DATA_BLOCK "DB_Z200_HMI"
{ DB_Accessible_From_OPC_UA := 'FALSE' ;
 DB_Accessible_From_Webserver := 'FALSE' ;
 S7_Optimized_Access := 'FALSE' }
VERSION : 0.1
NON_RETAIN
   STRUCT
      tALM { ExternalWritable := 'False'} : Struct   // HMI Alarms
         tE { ExternalWritable := 'False'} : Struct   // Emergency alarms
            xSpare_0 { ExternalWritable := 'False'} : Bool;
            xSpare_1 { ExternalWritable := 'False'} : Bool;
            xSpare_2 { ExternalWritable := 'False'} : Bool;
            xSpare_3 { ExternalWritable := 'False'} : Bool;
            xSpare_4 { ExternalWritable := 'False'} : Bool;
            xSpare_5 { ExternalWritable := 'False'} : Bool;
            xSpare_6 { ExternalWritable := 'False'} : Bool;
            xSpare_7 { ExternalWritable := 'False'} : Bool;
            xSpare_8 { ExternalWritable := 'False'} : Bool;
            xSpare_9 { ExternalWritable := 'False'} : Bool;
            xSpare_10 { ExternalWritable := 'False'} : Bool;
            xSpare_11 { ExternalWritable := 'False'} : Bool;
            xSpare_12 { ExternalWritable := 'False'} : Bool;
            xSpare_13 { ExternalWritable := 'False'} : Bool;
            xSpare_14 { ExternalWritable := 'False'} : Bool;
            xSpare_15 { ExternalWritable := 'False'} : Bool;
            xSpare_16 { ExternalWritable := 'False'} : Bool;
            xSpare_17 { ExternalWritable := 'False'} : Bool;
            xSpare_18 { ExternalWritable := 'False'} : Bool;
            xSpare_19 { ExternalWritable := 'False'} : Bool;
            xSpare_20 { ExternalWritable := 'False'} : Bool;
            xSpare_21 { ExternalWritable := 'False'} : Bool;
            xSpare_22 { ExternalWritable := 'False'} : Bool;
            xSpare_23 { ExternalWritable := 'False'} : Bool;
            xSpare_24 { ExternalWritable := 'False'} : Bool;
            xSpare_25 { ExternalWritable := 'False'} : Bool;
            xSpare_26 { ExternalWritable := 'False'} : Bool;
            xSpare_27 { ExternalWritable := 'False'} : Bool;
            xSpare_28 { ExternalWritable := 'False'} : Bool;
            xSpare_29 { ExternalWritable := 'False'} : Bool;
            xSpare_30 { ExternalWritable := 'False'} : Bool;
            xSpare_31 { ExternalWritable := 'False'} : Bool;
         END_STRUCT;
         tS { ExternalWritable := 'False'} : Struct   // Stopping faults
            xSpare_0 { ExternalWritable := 'False'} : Bool;   //
            xSpare_1 { ExternalWritable := 'False'} : Bool;
            xSpare_2 { ExternalWritable := 'False'} : Bool;
            xSpare_3 { ExternalWritable := 'False'} : Bool;
            xSpare_4 { ExternalWritable := 'False'} : Bool;
            xSpare_5 { ExternalWritable := 'False'} : Bool;
            xSpare_6 { ExternalWritable := 'False'} : Bool;
            xSpare_7 { ExternalWritable := 'False'} : Bool;
            xSpare_8 { ExternalWritable := 'False'} : Bool;
            xSpare_9 { ExternalWritable := 'False'} : Bool;
            xSpare_10 { ExternalWritable := 'False'} : Bool;
            xSpare_11 { ExternalWritable := 'False'} : Bool;
            xSpare_12 { ExternalWritable := 'False'} : Bool;
            xSpare_13 { ExternalWritable := 'False'} : Bool;
            xSpare_14 { ExternalWritable := 'False'} : Bool;
            xSpare_15 { ExternalWritable := 'False'} : Bool;
            xSpare_16 { ExternalWritable := 'False'} : Bool;
            xSpare_17 { ExternalWritable := 'False'} : Bool;
            xSpare_18 { ExternalWritable := 'False'} : Bool;
            xSpare_19 { ExternalWritable := 'False'} : Bool;
            xSpare_20 { ExternalWritable := 'False'} : Bool;
            xSpare_21 { ExternalWritable := 'False'} : Bool;
            xSpare_22 { ExternalWritable := 'False'} : Bool;
            xSpare_23 { ExternalWritable := 'False'} : Bool;
            xSpare_24 { ExternalWritable := 'False'} : Bool;
            xSpare_25 { ExternalWritable := 'False'} : Bool;
            xSpare_26 { ExternalWritable := 'False'} : Bool;
            xSpare_27 { ExternalWritable := 'False'} : Bool;
            xSpare_28 { ExternalWritable := 'False'} : Bool;
            xSpare_29 { ExternalWritable := 'False'} : Bool;
            xSpare_30 { ExternalWritable := 'False'} : Bool;
            xSpare_31 { ExternalWritable := 'False'} : Bool;
         END_STRUCT;
         tF { ExternalWritable := 'False'} : Struct   // Faults
            xSpare_0 { ExternalWritable := 'False'} : Bool;
            xProtectionCommandsAnomalies { ExternalWritable := 'False'} : Bool;   // R18QF3.Power supply 24v logic
            xProtectionInternalInputAnomalies { ExternalWritable := 'False'} : Bool;   // R18QF4.Power supply 24v logic
            xRedundancy24vOK1 { ExternalWritable := 'False'} : Bool;   // R18AP1.Redundancy 24v ok
            xProtectionInternalOutputAnomalies { ExternalWritable := 'False'} : Bool;   // R18QF7.Power supply 24v logic
            xProtectionExternalInputAnomalies { ExternalWritable := 'False'} : Bool;   // R18QF8.Power supply 24v logic
            xSpare_6 { ExternalWritable := 'False'} : Bool;   //
            xSpare_7 { ExternalWritable := 'False'} : Bool;
            xSpare_8 { ExternalWritable := 'False'} : Bool;   //
            xSpare_9 { ExternalWritable := 'False'} : Bool;
            xSpare_10 { ExternalWritable := 'False'} : Bool;   //
            xSpare_11 { ExternalWritable := 'False'} : Bool;
            xSpare_12 { ExternalWritable := 'False'} : Bool;
            xSpare_13 { ExternalWritable := 'False'} : Bool;
            xSpare_14 { ExternalWritable := 'False'} : Bool;
            xSpare_15 { ExternalWritable := 'False'} : Bool;
            xSpare_16 { ExternalWritable := 'False'} : Bool;
            xCompressedAirCutting { ExternalWritable := 'False'} : Bool;   // R427SP1.Compressed air presence cutting bridges
            xPowerSupply24v_R18QF5_CPU_A { ExternalWritable := 'False'} : Bool;   // R18QF5.Power supply 24v CPU A
            xPowerSupply24v_R18QF6_CPU_B { ExternalWritable := 'False'} : Bool;   // R18QF6.Power supply 24v CPU B
            xPowerSupply24vProt1 { ExternalWritable := 'False'} : Bool;
            xPowerSupply24vProt2 { ExternalWritable := 'False'} : Bool;
            xMissingCPU_A_abilitation { ExternalWritable := 'False'} : Bool;
            xMissingCPU_B_abilitation { ExternalWritable := 'False'} : Bool;
            xSpare_24 { ExternalAccessible := 'False'; ExternalVisible := 'False'; ExternalWritable := 'False'} : Bool;
            xSpare_25 { ExternalAccessible := 'False'; ExternalVisible := 'False'; ExternalWritable := 'False'} : Bool;
            xSpare_26 { ExternalAccessible := 'False'; ExternalVisible := 'False'; ExternalWritable := 'False'} : Bool;
            xSpare_27 { ExternalAccessible := 'False'; ExternalVisible := 'False'; ExternalWritable := 'False'} : Bool;
            xSpare_28 { ExternalAccessible := 'False'; ExternalVisible := 'False'; ExternalWritable := 'False'} : Bool;
            xSpare_29 { ExternalAccessible := 'False'; ExternalVisible := 'False'; ExternalWritable := 'False'} : Bool;
            xSpare_30 { ExternalAccessible := 'False'; ExternalVisible := 'False'; ExternalWritable := 'False'} : Bool;
            xSpare_31 { ExternalAccessible := 'False'; ExternalVisible := 'False'; ExternalWritable := 'False'} : Bool;
         END_STRUCT;
         tW { ExternalWritable := 'False'} : Struct   // Warnings
            xPowerFailure230vAux { ExternalWritable := 'False'} : Bool;   // R11QF2/3.Power failure 230v auxiliary
            xSpare_1 { ExternalWritable := 'False'} : Bool;
            xSpare_2 { ExternalWritable := 'False'} : Bool;
            xSpare_3 { ExternalWritable := 'False'} : Bool;
            xSpare_4 { ExternalWritable := 'False'} : Bool;
            xSpare_5 { ExternalWritable := 'False'} : Bool;
            xSpare_6 { ExternalWritable := 'False'} : Bool;
            xSpare_7 { ExternalWritable := 'False'} : Bool;
            xSpare_8 { ExternalWritable := 'False'} : Bool;
            xSpare_9 { ExternalWritable := 'False'} : Bool;
            xSpare_10 { ExternalWritable := 'False'} : Bool;
            xSpare_11 { ExternalWritable := 'False'} : Bool;
            xSpare_12 { ExternalWritable := 'False'} : Bool;
            xSpare_13 { ExternalWritable := 'False'} : Bool;
            xSpare_14 { ExternalWritable := 'False'} : Bool;
            xSpare_15 { ExternalWritable := 'False'} : Bool;
            xSpare_16 { ExternalWritable := 'False'} : Bool;
            xSpare_17 { ExternalWritable := 'False'} : Bool;
            xSpare_18 { ExternalWritable := 'False'} : Bool;
            xSpare_19 { ExternalWritable := 'False'} : Bool;
            xSpare_20 { ExternalWritable := 'False'} : Bool;
            xSpare_21 { ExternalWritable := 'False'} : Bool;
            xSpare_22 { ExternalWritable := 'False'} : Bool;
            xSpare_23 { ExternalWritable := 'False'} : Bool;
            xSpare_24 { ExternalWritable := 'False'} : Bool;
            xSpare_25 { ExternalWritable := 'False'} : Bool;
            xSpare_26 { ExternalWritable := 'False'} : Bool;
            xSpare_27 { ExternalWritable := 'False'} : Bool;
            xSpare_28 { ExternalWritable := 'False'} : Bool;
            xSpare_29 { ExternalWritable := 'False'} : Bool;
            xSpare_30 { ExternalWritable := 'False'} : Bool;
            xSpare_31 { ExternalWritable := 'False'} : Bool;
         END_STRUCT;
      END_STRUCT;
      tHMR { ExternalWritable := 'False'} : Struct   // HMI Read
         xSpare0 { ExternalWritable := 'False'} : Bool;
         xSpare1 { ExternalWritable := 'False'} : Bool;
         xSpare2 { ExternalWritable := 'False'} : Bool;
         xSpare3 { ExternalWritable := 'False'} : Bool;
         xSpare4 { ExternalWritable := 'False'} : Bool;
         xSpare5 { ExternalWritable := 'False'} : Bool;
         xSpare6 { ExternalWritable := 'False'} : Bool;
         xSpare7 { ExternalWritable := 'False'} : Bool;
         xSpare8 { ExternalWritable := 'False'} : Bool;
         xSpare9 { ExternalWritable := 'False'} : Bool;
         xSpare10 { ExternalWritable := 'False'} : Bool;
         xSpare11 { ExternalWritable := 'False'} : Bool;
         xSpare12 { ExternalWritable := 'False'} : Bool;
         xSpare13 { ExternalWritable := 'False'} : Bool;
         xSpare14 { ExternalWritable := 'False'} : Bool;
         xZoneAlarm { ExternalWritable := 'False'} : Bool;   // Zone alarm {X|X|X|X|O}
         xSpare16 { ExternalWritable := 'False'} : Bool;
         xSpare17 { ExternalWritable := 'False'} : Bool;
         xSpare18 { ExternalWritable := 'False'} : Bool;
         xSpare19 { ExternalWritable := 'False'} : Bool;
         xSpare20 { ExternalWritable := 'False'} : Bool;
         xSpare21 { ExternalWritable := 'False'} : Bool;
         xSpare22 { ExternalWritable := 'False'} : Bool;
         xSpare23 { ExternalWritable := 'False'} : Bool;
         xSpare24 { ExternalWritable := 'False'} : Bool;
         xSpare25 { ExternalWritable := 'False'} : Bool;
         xSpare26 { ExternalWritable := 'False'} : Bool;
         xSpare27 { ExternalWritable := 'False'} : Bool;
         xSpare28 { ExternalWritable := 'False'} : Bool;
         xSpare29 { ExternalWritable := 'False'} : Bool;
         xSpare30 { ExternalWritable := 'False'} : Bool;
         xSpare31 { ExternalWritable := 'False'} : Bool;
         xSpare { ExternalWritable := 'False'} : Array[0..15] of Bool;
         iSpare0 { ExternalWritable := 'False'} : Int;
         iSpare1 { ExternalWritable := 'False'} : Int;
         iSpare2 { ExternalWritable := 'False'} : Int;
         iSpare3 { ExternalWritable := 'False'} : Int;
         iSpare4 { ExternalWritable := 'False'} : Int;
         iSpare5 { ExternalWritable := 'False'} : Int;
         iSpare6 { ExternalWritable := 'False'} : Int;
         iSpare7 { ExternalWritable := 'False'} : Int;
         iSpare8 { ExternalWritable := 'False'} : Int;
         iSpare9 { ExternalWritable := 'False'} : Int;
         iSpare10 { ExternalWritable := 'False'} : Int;
         iSpare11 { ExternalWritable := 'False'} : Int;
         iSpare12 { ExternalWritable := 'False'} : Int;
         iSpare13 { ExternalWritable := 'False'} : Int;
         iSpare14 { ExternalWritable := 'False'} : Int;
         iSpare15 { ExternalWritable := 'False'} : Int;
         iSpare16 { ExternalWritable := 'False'} : Int;
         dSpare0 { ExternalWritable := 'False'} : DInt;
         dZoneState { ExternalWritable := 'False'} : DInt;   // Zone status (1=CycleON 2=StopCyc 4=CycleReq 8=StopReq 1024=E-Stop) {X|X|X|X|O}
         dCabinetStatusMCC1200 { ExternalWritable := 'False'} : DInt;   // Cabinet status MCC1200 (0=OK;1=General power alarm;2=Local power alarm) {X|X|X|X|O}
         dSpare3 { ExternalWritable := 'False'} : DInt;   //
         dSpare4 { ExternalWritable := 'False'} : DInt;
         dSpare5 { ExternalWritable := 'False'} : DInt;
         dSpare6 { ExternalWritable := 'False'} : DInt;
         dSpare7 { ExternalWritable := 'False'} : DInt;
         dSpare8 { ExternalWritable := 'False'} : DInt;
         dSpare9 { ExternalWritable := 'False'} : DInt;
         dSpare10 { ExternalWritable := 'False'} : DInt;
         dSpare11 { ExternalWritable := 'False'} : DInt;
         dSpare12 { ExternalWritable := 'False'} : DInt;
         dSpare13 { ExternalWritable := 'False'} : DInt;
         dSpare14 { ExternalWritable := 'False'} : DInt;
         dSpare15 { ExternalWritable := 'False'} : DInt;
         rSpare0 { ExternalWritable := 'False'} : Real;
         rSpare1 { ExternalWritable := 'False'} : Real;
         rSpare2 { ExternalWritable := 'False'} : Real;
         rSpare3 { ExternalWritable := 'False'} : Real;
         rSpare4 { ExternalWritable := 'False'} : Real;
         rSpare5 { ExternalWritable := 'False'} : Real;
         rSpare6 { ExternalWritable := 'False'} : Real;
         rSpare7 { ExternalWritable := 'False'} : Real;
         rSpare8 { ExternalWritable := 'False'} : Real;
         tManCmd { ExternalWritable := 'False'} : Struct
            xSpare0 { ExternalWritable := 'False'} : Bool;   //
            xSpare1 { ExternalWritable := 'False'} : Bool;
            xSpare2 { ExternalWritable := 'False'} : Bool;
            xSpare3 { ExternalWritable := 'False'} : Bool;
            xSpare4 { ExternalWritable := 'False'} : Bool;
            xSpare5 { ExternalWritable := 'False'} : Bool;
            xSpare6 { ExternalWritable := 'False'} : Bool;
            xSpare7 { ExternalWritable := 'False'} : Bool;
            xSpare8 { ExternalWritable := 'False'} : Bool;
            xSpare9 { ExternalWritable := 'False'} : Bool;
            xSpare10 { ExternalWritable := 'False'} : Bool;
            xSpare11 { ExternalWritable := 'False'} : Bool;
            xSpare12 { ExternalWritable := 'False'} : Bool;
            xSpare13 { ExternalWritable := 'False'} : Bool;
            xSpare14 { ExternalWritable := 'False'} : Bool;
            xSpare15 { ExternalWritable := 'False'} : Bool;
            xSpare { ExternalWritable := 'False'} : Array[0..15] of Bool;
         END_STRUCT;
      END_STRUCT;
      tHMW : Struct   // HMI Write
         xSpare0 : Bool;   //
         xSpare1 : Bool;
         xSpare2 : Bool;
         xSpare3 : Bool;
         xSpare4 : Bool;
         xSpare5 : Bool;
         xSpare6 : Bool;
         xSpare7 : Bool;
         xSpare8 : Bool;
         xSpare9 { ExternalWritable := 'False'} : Bool;
         xSpare10 : Bool;
         xSpare11 : Bool;
         xSpare12 : Bool;
         xSpare13 : Bool;
         xSpare14 : Bool;
         xSpare15 : Bool;
         xSpare16 : Bool;
         xSpare17 : Bool;
         xSpare18 : Bool;
         xSpare19 : Bool;
         xSpare20 : Bool;
         xSpare21 : Bool;
         xSpare22 : Bool;
         xSpare23 : Bool;
         xSpare24 : Bool;
         xSpare25 : Bool;
         xSpare26 : Bool;
         xSpare27 : Bool;
         xSpare28 : Bool;
         xSpare29 : Bool;
         xSpare30 : Bool;
         xSpare31 : Bool;
         xSpare : Array[0..15] of Bool;
         iSpare0 : Int;
         iSpare1 : Int;
         iSpare2 : Int;
         iSpare3 : Int;
         iSpare4 : Int;
         iSpare5 : Int;
         iSpare6 : Int;
         iSpare7 : Int;
         iSpare8 : Int;
         iSpare9 : Int;
         iSpare10 : Int;
         iSpare11 : Int;
         iSpare12 : Int;
         iSpare13 : Int;
         iSpare14 : Int;
         iSpare15 : Int;
         iSpare16 : Int;
         dSpare0 : DInt;
         dSpare1 : DInt;
         dSpare2 : DInt;   //
         dSpare3 : DInt;
         dSpare4 : DInt;
         dSpare5 : DInt;
         dSpare6 : DInt;
         dSpare7 : DInt;
         dSpare8 : DInt;
         dSpare9 : DInt;
         dSpare10 : DInt;
         dSpare11 : DInt;
         dSpare12 : DInt;
         dSpare13 : DInt;
         dSpare14 : DInt;
         dSpare15 : DInt;
         dSpare16 : DInt;
         rSpare0 : Real;
         rSpare1 : Real;
         rSpare2 : Real;
         rSpare3 : Real;
         rSpare4 : Real;
         rSpare5 : Real;
         rSpare6 : Real;
         rSpare7 : Real;
         rSpare8 : Real;
         tManCmd : Struct
            xSpare0 : Bool;
            xSpare1 : Bool;
            xSpare2 { ExternalWritable := 'False'} : Bool;
            xSpare3 { ExternalWritable := 'False'} : Bool;
            xSpare4 { ExternalWritable := 'False'} : Bool;
            xSpare5 { ExternalWritable := 'False'} : Bool;
            xSpare6 { ExternalWritable := 'False'} : Bool;
            xSpare7 { ExternalWritable := 'False'} : Bool;
            xSpare8 { ExternalWritable := 'False'} : Bool;
            xSpare9 { ExternalWritable := 'False'} : Bool;
            xSpare10 { ExternalWritable := 'False'} : Bool;
            xSpare11 { ExternalWritable := 'False'} : Bool;
            xSpare12 { ExternalWritable := 'False'} : Bool;
            xSpare13 { ExternalWritable := 'False'} : Bool;
            xSpare14 { ExternalWritable := 'False'} : Bool;
            xSpare15 { ExternalWritable := 'False'} : Bool;
            xSpare16 : Bool;
            xSpare17 : Bool;
            xSpare18 : Bool;
            xSpare19 : Bool;
            xSpare20 : Bool;
            xSpare21 : Bool;
            xSpare22 : Bool;
            xSpare23 : Bool;
            xSpare24 : Bool;
            xSpare25 : Bool;
            xSpare26 : Bool;
            xSpare27 : Bool;
            xSpare28 : Bool;
            xSpare29 : Bool;
            xSpare30 : Bool;
            xSpare31 : Bool;
         END_STRUCT;
      END_STRUCT;
   END_STRUCT;


BEGIN
   tALM.tE.xSpare_0 := FALSE;
   tALM.tE.xSpare_1 := FALSE;
   tALM.tE.xSpare_2 := FALSE;
   tALM.tE.xSpare_3 := FALSE;
   tALM.tE.xSpare_4 := FALSE;
   tALM.tE.xSpare_5 := FALSE;
   tALM.tE.xSpare_6 := FALSE;
   tALM.tE.xSpare_7 := FALSE;
   tALM.tE.xSpare_8 := FALSE;
   tALM.tE.xSpare_9 := FALSE;
   tALM.tE.xSpare_10 := FALSE;
   tALM.tE.xSpare_11 := FALSE;
   tALM.tE.xSpare_12 := FALSE;
   tALM.tE.xSpare_13 := FALSE;
   tALM.tE.xSpare_14 := FALSE;
   tALM.tE.xSpare_15 := FALSE;
   tALM.tE.xSpare_16 := FALSE;
   tALM.tE.xSpare_17 := FALSE;
   tALM.tE.xSpare_18 := FALSE;
   tALM.tE.xSpare_19 := FALSE;
   tALM.tE.xSpare_20 := FALSE;
   tALM.tE.xSpare_21 := FALSE;
   tALM.tE.xSpare_22 := FALSE;
   tALM.tE.xSpare_23 := FALSE;
   tALM.tE.xSpare_24 := FALSE;
   tALM.tE.xSpare_25 := FALSE;
   tALM.tE.xSpare_26 := FALSE;
   tALM.tE.xSpare_27 := FALSE;
   tALM.tE.xSpare_28 := FALSE;
   tALM.tE.xSpare_29 := FALSE;
   tALM.tE.xSpare_30 := FALSE;
   tALM.tE.xSpare_31 := FALSE;
   tALM.tS.xSpare_0 := FALSE;
   tALM.tS.xSpare_1 := FALSE;
   tALM.tS.xSpare_2 := FALSE;
   tALM.tS.xSpare_3 := FALSE;
   tALM.tS.xSpare_4 := FALSE;
   tALM.tS.xSpare_5 := FALSE;
   tALM.tS.xSpare_6 := FALSE;
   tALM.tS.xSpare_7 := FALSE;
   tALM.tS.xSpare_8 := FALSE;
   tALM.tS.xSpare_9 := FALSE;
   tALM.tS.xSpare_10 := FALSE;
   tALM.tS.xSpare_11 := FALSE;
   tALM.tS.xSpare_12 := FALSE;
   tALM.tS.xSpare_13 := FALSE;
   tALM.tS.xSpare_14 := FALSE;
   tALM.tS.xSpare_15 := FALSE;
   tALM.tS.xSpare_16 := FALSE;
   tALM.tS.xSpare_17 := FALSE;
   tALM.tS.xSpare_18 := FALSE;
   tALM.tS.xSpare_19 := FALSE;
   tALM.tS.xSpare_20 := FALSE;
   tALM.tS.xSpare_21 := FALSE;
   tALM.tS.xSpare_22 := FALSE;
   tALM.tS.xSpare_23 := FALSE;
   tALM.tS.xSpare_24 := FALSE;
   tALM.tS.xSpare_25 := FALSE;
   tALM.tS.xSpare_26 := FALSE;
   tALM.tS.xSpare_27 := FALSE;
   tALM.tS.xSpare_28 := FALSE;
   tALM.tS.xSpare_29 := FALSE;
   tALM.tS.xSpare_30 := FALSE;
   tALM.tS.xSpare_31 := FALSE;
   tALM.tF.xSpare_0 := TRUE;
   tALM.tF.xProtectionCommandsAnomalies := FALSE;
   tALM.tF.xProtectionInternalInputAnomalies := FALSE;
   tALM.tF.xRedundancy24vOK1 := FALSE;
   tALM.tF.xProtectionInternalOutputAnomalies := FALSE;
   tALM.tF.xProtectionExternalInputAnomalies := FALSE;
   tALM.tF.xSpare_6 := FALSE;
   tALM.tF.xSpare_7 := FALSE;
   tALM.tF.xSpare_8 := FALSE;
   tALM.tF.xSpare_9 := FALSE;
   tALM.tF.xSpare_10 := FALSE;
   tALM.tF.xSpare_11 := FALSE;
   tALM.tF.xPowerSupply24vProt1 := FALSE;
   tALM.tF.xPowerSupply24vProt2 := FALSE;
   tALM.tF.xMissingCPU_A_abilitation := FALSE;
   tALM.tF.xMissingCPU_B_abilitation := FALSE;
   tALM.tF.xSpare_24 := FALSE;
   tALM.tF.xSpare_25 := FALSE;
   tALM.tF.xSpare_26 := FALSE;
   tALM.tF.xSpare_27 := FALSE;
   tALM.tF.xSpare_28 := FALSE;
   tALM.tF.xSpare_29 := FALSE;
   tALM.tF.xSpare_30 := FALSE;
   tALM.tF.xSpare_31 := FALSE;
   tALM.tW.xPowerFailure230vAux := FALSE;
   tALM.tW.xSpare_1 := FALSE;
   tALM.tW.xSpare_2 := FALSE;
   tALM.tW.xSpare_3 := FALSE;
   tALM.tW.xSpare_4 := FALSE;
   tALM.tW.xSpare_5 := FALSE;
   tALM.tW.xSpare_6 := FALSE;
   tALM.tW.xSpare_7 := FALSE;
   tALM.tW.xSpare_8 := FALSE;
   tALM.tW.xSpare_9 := FALSE;
   tALM.tW.xSpare_10 := FALSE;
   tALM.tW.xSpare_11 := FALSE;
   tALM.tW.xSpare_12 := FALSE;
   tALM.tW.xSpare_13 := FALSE;
   tALM.tW.xSpare_14 := FALSE;
   tALM.tW.xSpare_15 := FALSE;
   tALM.tW.xSpare_16 := FALSE;
   tALM.tW.xSpare_17 := FALSE;
   tALM.tW.xSpare_18 := FALSE;
   tALM.tW.xSpare_19 := FALSE;
   tALM.tW.xSpare_20 := FALSE;
   tALM.tW.xSpare_21 := FALSE;
   tALM.tW.xSpare_22 := FALSE;
   tALM.tW.xSpare_23 := FALSE;
   tALM.tW.xSpare_24 := FALSE;
   tALM.tW.xSpare_25 := FALSE;
   tALM.tW.xSpare_26 := FALSE;
   tALM.tW.xSpare_27 := FALSE;
   tALM.tW.xSpare_28 := FALSE;
   tALM.tW.xSpare_29 := FALSE;
   tALM.tW.xSpare_30 := FALSE;
   tALM.tW.xSpare_31 := FALSE;
   tHMR.xZoneAlarm := FALSE;
   tHMR.dZoneState := 1024;
   tHMR.dCabinetStatusMCC1200 := 1;
   tHMW.xSpare5 := FALSE;
   tHMW.xSpare6 := FALSE;
   tHMW.xSpare7 := FALSE;
   tHMW.xSpare15 := FALSE;
   tHMW.xSpare16 := FALSE;

END_DATA_BLOCK

